// Mitsubishi GX Works2 project: infinite2   PLC: Q03UDV

PROGRAM MAIN
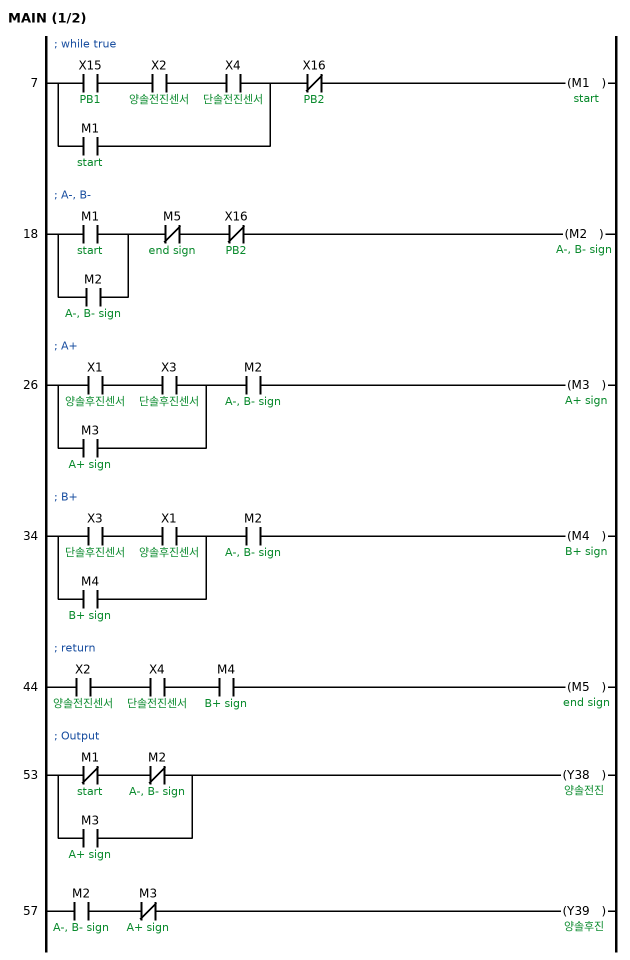
; while true
7     LD      X15  ; PB1
      AND     X2  ; 양솔전진센서
      AND     X4  ; 단솔전진센서
      OR      M1  ; start
      ANI     X16  ; PB2
      OUT     M1  ; start
; A-, B-
18    LD      M1  ; start
      OR      M2  ; A-, B- sign
      ANI     M5  ; end sign
      ANI     X16  ; PB2
      OUT     M2  ; A-, B- sign
; A+
26    LD      X1  ; 양솔후진센서
      AND     X3  ; 단솔후진센서
      OR      M3  ; A+ sign
      AND     M2  ; A-, B- sign
      OUT     M3  ; A+ sign
; B+
34    LD      X3  ; 단솔후진센서
      AND     X1  ; 양솔후진센서
      OR      M4  ; B+ sign
      AND     M2  ; A-, B- sign
      OUT     M4  ; B+ sign
; return
44    LD      X2  ; 양솔전진센서
      AND     X4  ; 단솔전진센서
      AND     M4  ; B+ sign
      OUT     M5  ; end sign
; Output
53    LDI     M1  ; start
      ANI     M2  ; A-, B- sign
      OR      M3  ; A+ sign
      OUT     Y38  ; 양솔전진
57    LD      M2  ; A-, B- sign
      ANI     M3  ; A+ sign
      OUT     Y39  ; 양솔후진
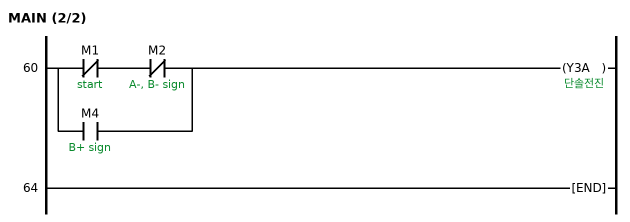
60    LDI     M1  ; start
      ANI     M2  ; A-, B- sign
      OR      M4  ; B+ sign
      OUT     Y3A  ; 단솔전진
64    END
END_PROGRAM

// device comments not shown above
M6  ; end sign
